FUNCTION_BLOCK LightSensor (* Basic Function Block Type *)
  (* Standard: 61499-2 *)
  (* Version 0.0, 21/06/2022, Lernfabrik, WBK hackaton, Template *)
  PACKAGE Main;
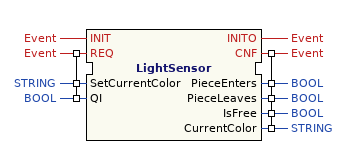
  EVENT_INPUT
    INIT; (* Initialization Request *)
    REQ WITH SetCurrentColor, QI; (* Normal Execution Request *)
  END_EVENT
  EVENT_OUTPUT
    INITO; (* Initialization Confirm *)
    CNF WITH PieceEnters, PieceLeaves, IsFree, CurrentColor; (* Execution Confirmation *)
  END_EVENT
  VAR_INPUT
    SetCurrentColor : STRING;
    QI : BOOL;
  END_VAR
  VAR_OUTPUT
    PieceEnters : BOOL;
    PieceLeaves : BOOL;
    IsFree : BOOL;
    CurrentColor : STRING;
  END_VAR
  VAR
    CurrentPiecesColor : STRING;
    PieceIsIn : BOOL;
  END_VAR
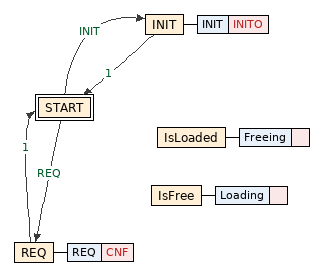
  EC_STATES
    START; (* Initial State *)
    INIT : INIT -> INITO; (* Initialization *)
    REQ : REQ -> CNF; (* Normal execution *)
    IsFree : Loading;
    IsLoaded : Freeing;
  END_STATES
  EC_TRANSITIONS
    START TO INIT := INIT;
    INIT TO START := 1;
    START TO REQ := REQ;
    REQ TO START := 1;
  END_TRANSITIONS
  ALGORITHM INIT IN ST: (* Initialization algorithm *)
;
  END_ALGORITHM
  ALGORITHM REQ IN ST: (* Normally executed algorithm *)
IF IsFree = TRUE AND QI = FALSE THEN
	PieceEnters := TRUE;
	IsFree := FALSE;
	PieceLeaves := FALSE;
ELSIF IsFree = FALSE AND QI = TRUE THEN
	PieceEnters := FALSE;
	IsFree := TRUE;
	PieceLeaves := TRUE;
ELSIF IsFree = TRUE AND QI = FALSE THEN
	IsFree := TRUE;
	PieceLeaves := FALSE;
	PieceEnters := FALSE;
ELSIF IsFree = FALSE AND QI = TRUE THEN
	IsFree := FALSE;
	PieceLeaves := FALSE;
	PieceEnters := FALSE;
END_IF;

IF SetCurrentColor <> '' THEN
	CurrentColor := SetCurrentColor;
	END_IF;
  END_ALGORITHM
  ALGORITHM Freeing IN ST:
;
  END_ALGORITHM
  ALGORITHM Loading IN ST:
;
  END_ALGORITHM
END_FUNCTION_BLOCK
